TYPE MNG_APPLICATION_INPUTS_32BIT :
STRUCT
    NumSignals                     : INT     := 1         ;
    init_sensor_creme_beckhoff_module_IR : BOOL    := 0; (* modul_Beckhoff/init_sensor_creme_beckhoff_module?IR *)
END_STRUCT
END_TYPE

(* stored: Version 1.1.0.1, ProductVersion 3.1.0.23 *)
